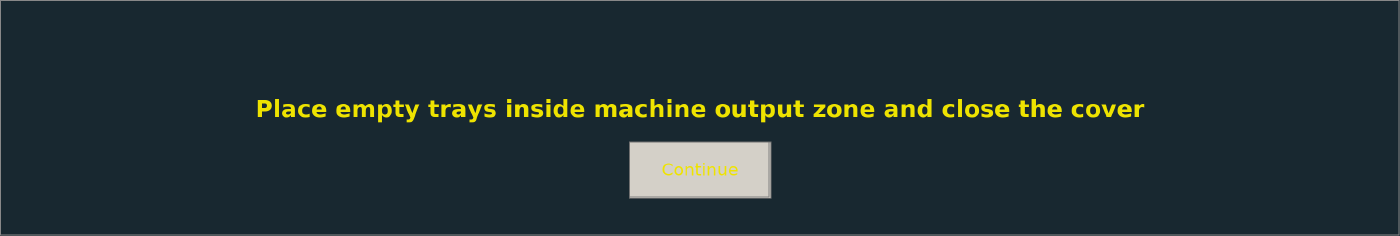
VISUALIZATION InitializingRotaryTablePlaceTrayDialog  // 1480x250
VAR_IN_OUT
	stInitializationRotaryTableFrame : ST_InitializationRotaryTableFrame;
END_VAR
    Label (0,95 1480x40), "Place empty trays inside machine output zone and close the cover"
    Button (665,150 150x60), "Continue", input disabled if: stInitializationRotaryTableFrame.bContinueDisabled
        toggle stInitializationRotaryTableFrame.btnContinue
END_VISUALIZATION

(* stored: Version 1.1.0.1, ProductVersion 3.1.4024.9
   Visu InitializingRotaryTablePlaceTrayDialog: Id {d516c153-6730-4bdb-9bc6-070a062e3b4a} *)
